PROGRAM prgReadWrite
VAR
	fbRW		: FB_ReadWrite;
END_VAR

fbRW(bBusy=> , bError=> , udiErrorCodeOut=> , eErrorReadWrite_Out=> );

END_PROGRAM

(* stored: Version 1.1.0.1, ProductVersion 3.1.4024.11
   POU prgReadWrite: Id {01d06878-4e44-4b4a-808b-89cc4c311023}, SpecialFunc None *)
